Staubli VAL3: JointStateMsg.pjx

Parameters version=s7.7.2 stackSize=5000 millimeterUnit=true
Program file=start.pgx
Program file=stop.pgx
Data file=JointStateMsg.dtx
Type name=Body path=../Body/Body.pjx
Type name=Prefix path=../Prefix/Prefix.pjx
Type name=Header path=../Header/Header.pjx
Type name=JointState path=../JointState/JointState.pjx
